{attribute 'qualified_only'}
{attribute 'strict'}
TYPE E_HMI_CONTROL_REQUEST :
(
	Default,
	RecipeMgmtRequest,
	SettingMgmtRequest,
	UserMgmtRequest
);   	
END_TYPE

(* stored: Version 1.1.0.1, ProductVersion 3.1.4024.11
   DUT E_HMI_CONTROL_REQUEST: Id {42c54a19-ecfd-4883-a64d-3f2be5338dc3} *)
